PROGRAM FunctionsAndFunctionBlocksex01
VAR
number1 		: number;
number2			: number;
sum12			: number;
END_VAR

number1 + number2 := sum12;

END_PROGRAM

(* stored: Version 1.1.0.1
   POU FunctionsAndFunctionBlocksex01: Id {405b5233-a6ad-494c-9ade-7bfcc71bf94f}, SpecialFunc None *)
